FUNCTION_BLOCK xaxpy
VAR_INPUT
    b_n: DINT;
    a: LREAL;
    ix0: DINT;
    iy0: DINT;
END_VAR
VAR_IN_OUT
    y: ARRAY [0..29] OF LREAL;
END_VAR
VAR_TEMP
    ix: DINT;
    iy: DINT;
    k: DINT;
END_VAR

IF (b_n >= 1) AND (a <> 0.0) THEN 
    ix := ix0 - 1;
    iy := iy0 - 1;
    k := 0;
    WHILE k <= (b_n - 1) DO
        y[iy] := (a * y[ix]) + y[iy];
        ix := ix + 1;
        iy := iy + 1;
        k := k + 1;
    END_WHILE;
END_IF;

END_FUNCTION_BLOCK

(* stored: Version 1.1.0.1, ProductVersion 3.1.4024.12
   POU xaxpy: Id {3f1b4712-e214-4eb0-aa41-495a3e54ec9d}, SpecialFunc None *)
